TYPE EtcMasterBase_62654B43 :
STRUCT
END_STRUCT
END_TYPE

(* stored: Version 1.2.0.0, ProductVersion 3.1.4024.9
   DUT EtcMasterBase_62654B43: Id {53ff24cc-20d3-413b-bf55-fc1dadf94fee} *)
